(* Schneider Machine Expert - Basic project MES_I40, file version 2.8.0.0 *)
(* CompanyInformations: Name=BAZZICA *)
(* ProjectInformations: Name=Mulino Bazzica *)
(* UserInformations: LastName=Dominici, FirstName=Erica, PhoneNumber=+39 0742 38501, Email=info@promas.com, Street=via XXV Aprile, 10/12, City=Trevi, ZipCode=06039, State=Perugia, Country=Italy *)

HARDWARE
  Cpu 0: TM221CE16T
  Cartridge1 0: TMC2TI2
  EthernetConfiguration: NetworkName=M221, IpAllocationMode=FixedAddress, IpAddress=192.168.0.160, SubnetMask=255.255.254.0
  EthernetConfiguration: NetworkName=M221, IpAllocationMode=FixedAddress, IpAddress=0.0.0.0, SubnetMask=0.0.0.0
  SerialLineConfiguration: Baud=Baud19200, Parity=ParityEven, DataBits=DataBits8, StopBits=StopBits1, PhysicalMedium=PhysicalMediumRs485, TransmissionMode=TransmissionModeModbusRtu, SlaveId=1, Addressing=SlaveAddressing
  MastTask: UsePeriodScanMode=true, PeriodScan=100
  FastTask: Period=255
  CpuBehavior: StartingMode=StartInRun, AutoSaveRamOnEeprom=true, WatchdogPeriod=250

SYMBOLS  (address, symbol, comment, settings)
  %M0       NEW_CYCLE_TRIGGER_V
  %MW0        "LIFECYCLE COUNTER 1st WORD"
  %MW1      CYCLES_CNT_W1  "LIFECYCEL COUNTER 2nd WORD"
  %MW6      HMI_IN  "HMI_IN"
  %MW7      HMI_OUT  "DATA >> HMI"
  %MD0      CYCLES_CNT_W0
  %TM0      NEW_CYCLE_TRIGGER  [Preset=2, Base=OneSecond]
  %TM2        [Preset=3, Base=OneSecond]
  %TM3        [Preset=3, Base=OneSecond]
  %TM4        [Preset=3, Base=OneSecond]
  %TM5        [Preset=3, Base=OneSecond]
  %TM6        [Preset=3, Base=OneSecond]
  %TM7        [Preset=3, Base=OneSecond]
  %C0       LIFE_CYCLE_00  "CYCLE COUNTER"  [Preset=0]
  %C1       LIFE_CYCLE_01
  %I0.0     RUN  "MAC GENERAL RELAY ON"
  %I0.1     ALARM  "ALARM"
  %I0.2     MOLD_CHG  "MOLD CHANGE"
  %I0.3     MAN_AUTO  "MACHINE MODE MAN/AUT[1/0]"
  %I0.4     NEW_CYCLE  "NEW CYCLE TRIGGER (AT LOADING)"
  %I0.5     COMMIT_END  "MACHINE REACHED COMMIT TARGET"
  %I0.6       "SPARE"
  %I0.7       "SPARE"
  %I0.8       "SPARE"
  %Q0.0     REMOTE_STOP  "REMOTE STOP"
  %Q0.1     REMOTE_LOAD  "REMOTE RECIPE LOAD CMD"
  %Q0.2     SPARE_02
  %Q0.3     SPARE_03
  %Q0.4     SPARE_04
  %Q0.5     SPARE_05
  %Q0.6     SPARE_06
  %IW0.0      "M_PRESSURE"  [Type=Type_0_10V, Scope=Scope_Normal, Minimum=0, Maximum=1000]
  %IW0.1      "F_PRESSURE"  [Type=Type_0_10V, Scope=Scope_Normal, Minimum=0, Maximum=1000]
  %IW0.100    "M_TEMPERATURE"  [Type=Type_ThermocoupleK, Scope=Scope_Celsius, Minimum=-2000, Maximum=13000]
  %IW0.101    "F_TEMPERATURE"  [Type=Type_ThermocoupleK, Scope=Scope_Celsius, Minimum=-2000, Maximum=13000]

POU IN
  (* SectionNumber=1 *)

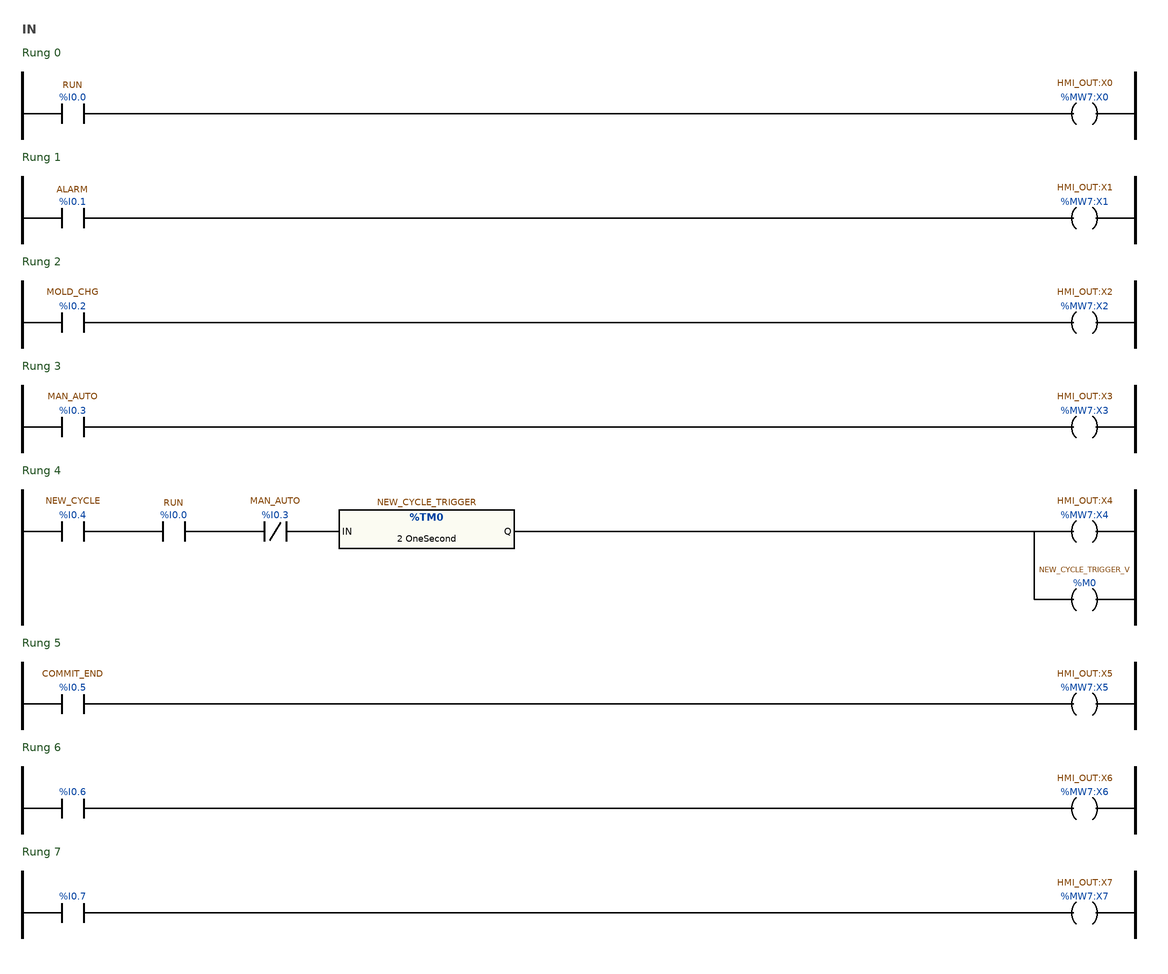

// Rung 0
  LD %I0.0                (* RUN *)
  ST %MW7:X0              (* HMI_OUT *)
  // as ST:
  //   HMI_OUT:X0 := RUN;

// Rung 1
  LD %I0.1                (* ALARM *)
  ST %MW7:X1              (* HMI_OUT *)
  // as ST:
  //   HMI_OUT:X1 := ALARM;

// Rung 2
  LD %I0.2                (* MOLD_CHG *)
  ST %MW7:X2              (* HMI_OUT *)
  // as ST:
  //   HMI_OUT:X2 := MOLD_CHG;

// Rung 3
  LD %I0.3                (* MAN_AUTO *)
  ST %MW7:X3              (* HMI_OUT *)
  // as ST:
  //   HMI_OUT:X3 := MAN_AUTO;

// Rung 4
  BLK %TM0                (* NEW_CYCLE_TRIGGER *)
  LD %I0.4                (* NEW_CYCLE *)
  AND %I0.0               (* RUN *)
  ANDN %I0.3              (* MAN_AUTO *)
  IN
  OUT_BLK
  LD Q
  ST %MW7:X4              (* HMI_OUT *)
  ST %M0                  (* NEW_CYCLE_TRIGGER_V *)
  END_BLK
  // as ST:
  //   NEW_CYCLE_TRIGGER(IN := NEW_CYCLE AND RUN AND NOT MAN_AUTO);
  //   HMI_OUT:X4 := NEW_CYCLE_TRIGGER.Q;
  //   NEW_CYCLE_TRIGGER_V := NEW_CYCLE_TRIGGER.Q;

// Rung 5
  LD %I0.5                (* COMMIT_END *)
  ST %MW7:X5              (* HMI_OUT *)
  // as ST:
  //   HMI_OUT:X5 := COMMIT_END;

// Rung 6
  LD %I0.6
  ST %MW7:X6              (* HMI_OUT *)
  // as ST:
  //   HMI_OUT:X6 := %I0.6;

// Rung 7
  LD %I0.7
  ST %MW7:X7              (* HMI_OUT *)
  // as ST:
  //   HMI_OUT:X7 := %I0.7;

POU TMR_CNT
  (* SectionNumber=2 *)

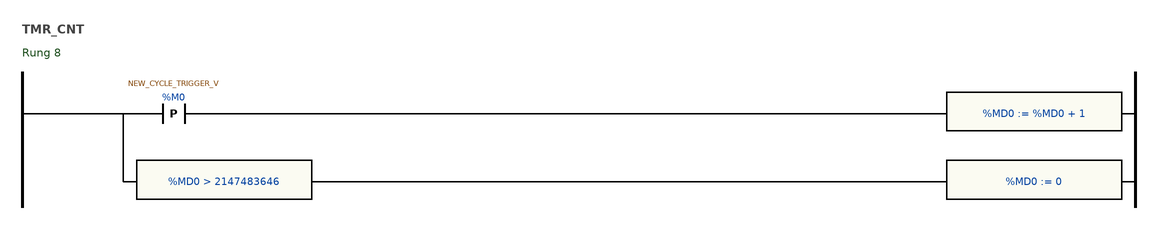

// Rung 8
  LD 1
  MPS
  ANDR %M0                (* NEW_CYCLE_TRIGGER_V *)
  [ %MD0 := %MD0 + 1 ]    (* CYCLES_CNT_W0, CYCLES_CNT_W0 *)
  MPP
  AND [ %MD0 > 2147483646 ](* CYCLES_CNT_W0 *)
  [ %MD0 := 0 ]           (* CYCLES_CNT_W0 *)
  // as ST:
  //   IF RISING(NEW_CYCLE_TRIGGER_V) THEN CYCLES_CNT_W0 := CYCLES_CNT_W0 + 1; END_IF;
  //   IF CYCLES_CNT_W0 > 2147483646 THEN CYCLES_CNT_W0 := 0; END_IF;

POU OUT
  (* SectionNumber=3 *)

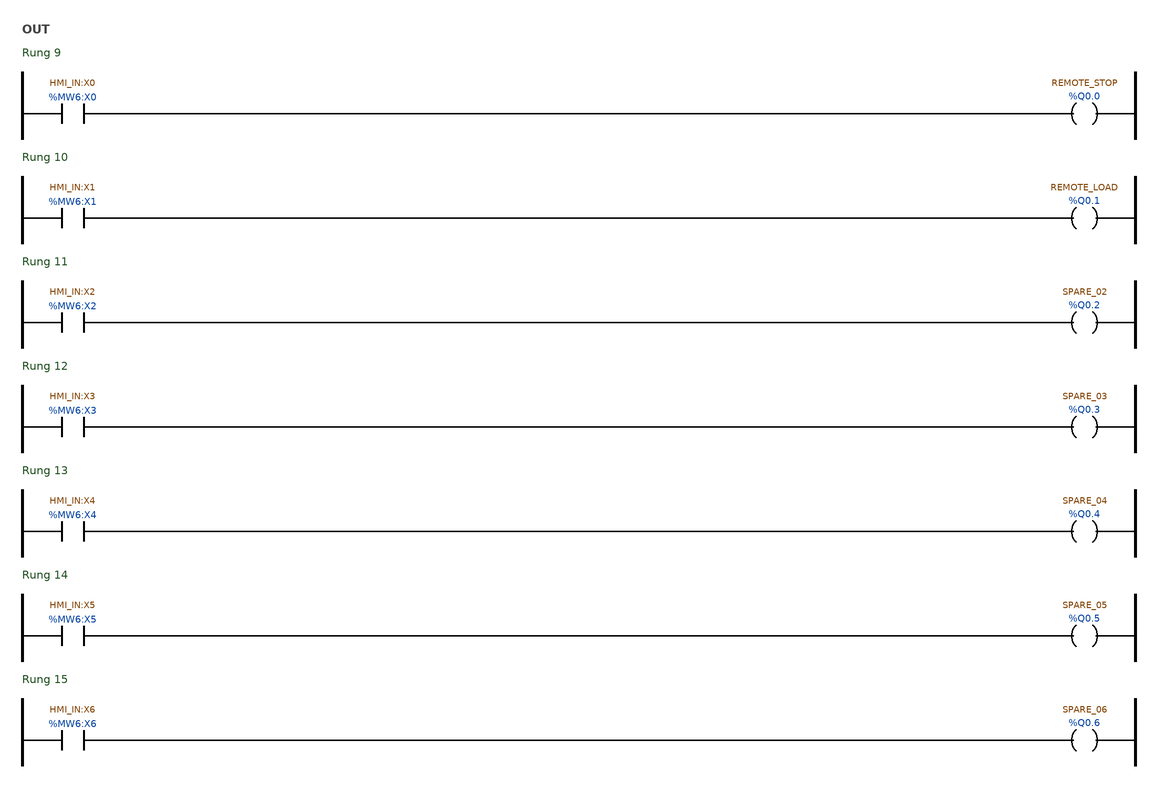

// Rung 9
  LD %MW6:X0              (* HMI_IN *)
  ST %Q0.0                (* REMOTE_STOP *)
  // as ST:
  //   REMOTE_STOP := HMI_IN:X0;

// Rung 10
  LD %MW6:X1              (* HMI_IN *)
  ST %Q0.1                (* REMOTE_LOAD *)
  // as ST:
  //   REMOTE_LOAD := HMI_IN:X1;

// Rung 11
  LD %MW6:X2              (* HMI_IN *)
  ST %Q0.2                (* SPARE_02 *)
  // as ST:
  //   SPARE_02 := HMI_IN:X2;

// Rung 12
  LD %MW6:X3              (* HMI_IN *)
  ST %Q0.3                (* SPARE_03 *)
  // as ST:
  //   SPARE_03 := HMI_IN:X3;

// Rung 13
  LD %MW6:X4              (* HMI_IN *)
  ST %Q0.4                (* SPARE_04 *)
  // as ST:
  //   SPARE_04 := HMI_IN:X4;

// Rung 14
  LD %MW6:X5              (* HMI_IN *)
  ST %Q0.5                (* SPARE_05 *)
  // as ST:
  //   SPARE_05 := HMI_IN:X5;

// Rung 15
  LD %MW6:X6              (* HMI_IN *)
  ST %Q0.6                (* SPARE_06 *)
  // as ST:
  //   SPARE_06 := HMI_IN:X6;

POU ALARMS
  (* SectionNumber=4 *)

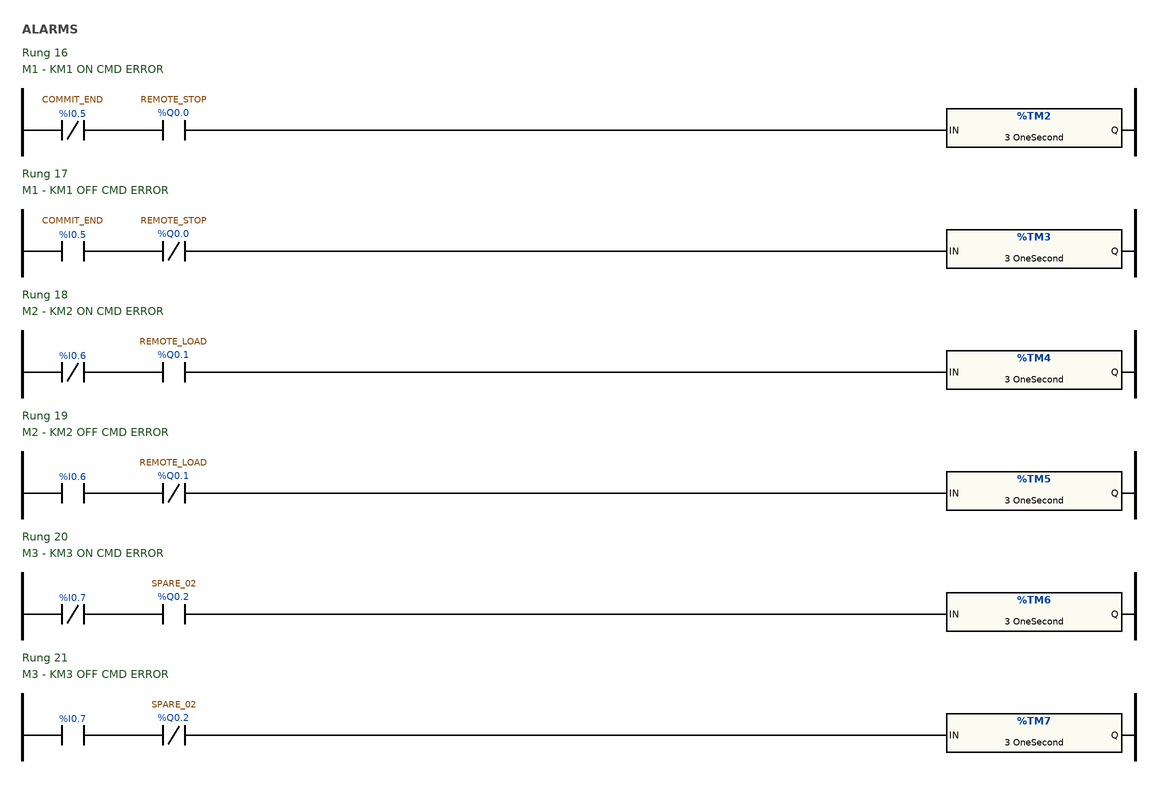

// Rung 16
// M1 - KM1 ON CMD ERROR
  BLK %TM2
  LDN %I0.5               (* COMMIT_END *)
  AND %Q0.0               (* REMOTE_STOP *)
  IN
  END_BLK
  // as ST:
  //   %TM2(IN := NOT COMMIT_END AND REMOTE_STOP);

// Rung 17
// M1 - KM1 OFF CMD ERROR
  BLK %TM3
  LD %I0.5                (* COMMIT_END *)
  ANDN %Q0.0              (* REMOTE_STOP *)
  IN
  END_BLK
  // as ST:
  //   %TM3(IN := COMMIT_END AND NOT REMOTE_STOP);

// Rung 18
// M2 - KM2 ON CMD ERROR
  BLK %TM4
  LDN %I0.6
  AND %Q0.1               (* REMOTE_LOAD *)
  IN
  END_BLK
  // as ST:
  //   %TM4(IN := NOT %I0.6 AND REMOTE_LOAD);

// Rung 19
// M2 - KM2 OFF CMD ERROR
  BLK %TM5
  LD %I0.6
  ANDN %Q0.1              (* REMOTE_LOAD *)
  IN
  END_BLK
  // as ST:
  //   %TM5(IN := %I0.6 AND NOT REMOTE_LOAD);

// Rung 20
// M3 - KM3 ON CMD ERROR
  BLK %TM6
  LDN %I0.7
  AND %Q0.2               (* SPARE_02 *)
  IN
  END_BLK
  // as ST:
  //   %TM6(IN := NOT %I0.7 AND SPARE_02);

// Rung 21
// M3 - KM3 OFF CMD ERROR
  BLK %TM7
  LD %I0.7
  ANDN %Q0.2              (* SPARE_02 *)
  IN
  END_BLK
  // as ST:
  //   %TM7(IN := %I0.7 AND NOT SPARE_02);

POU CONNECTION
  (* SectionNumber=5 *)

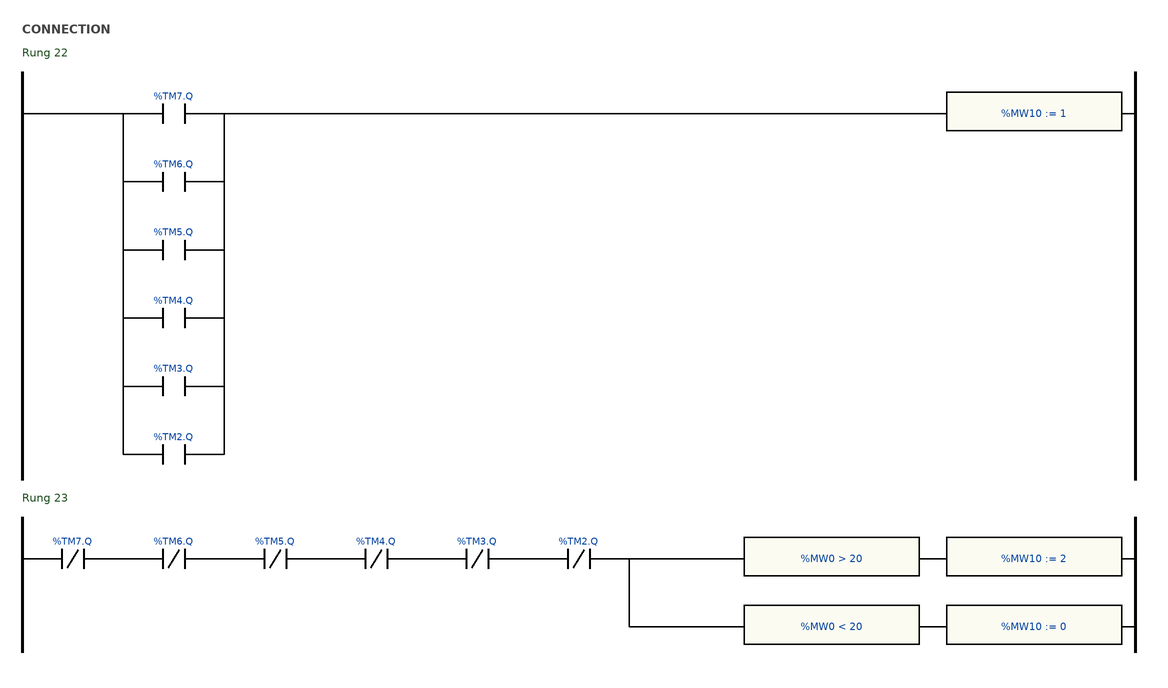

// Rung 22
  LD 1
  AND( %TM7.Q
  OR %TM6.Q
  OR %TM5.Q
  OR %TM4.Q
  OR %TM3.Q
  OR %TM2.Q
  )
  [ %MW10 := 1 ]
  // as ST:
  //   IF %TM7.Q OR %TM6.Q OR %TM5.Q OR %TM4.Q OR %TM3.Q OR %TM2.Q THEN %MW10 := 1; END_IF;

// Rung 23
  LDN %TM7.Q
  ANDN %TM6.Q
  ANDN %TM5.Q
  ANDN %TM4.Q
  ANDN %TM3.Q
  ANDN %TM2.Q
  MPS
  AND [ %MW0 > 20 ]
  [ %MW10 := 2 ]
  MPP
  AND [ %MW0 < 20 ]
  [ %MW10 := 0 ]
  // as ST:
  //   IF NOT %TM7.Q AND NOT %TM6.Q AND NOT %TM5.Q AND NOT %TM4.Q AND NOT %TM3.Q AND NOT %TM2.Q AND %MW0 > 20 THEN %MW10 := 2; END_IF;
  //   IF NOT %TM7.Q AND NOT %TM6.Q AND NOT %TM5.Q AND NOT %TM4.Q AND NOT %TM3.Q AND NOT %TM2.Q AND %MW0 < 20 THEN %MW10 := 0; END_IF;
